// TIA Portal V18 export
FUNCTION "Operator message 2" : Void   // FC33, LAD
{ S7_Optimized_Access := 'TRUE' }
VERSION : 0.1
// stored: AutoNumber true, IsIECCheckEnabled false, SetENOAutomatically false, UDAEnableTagReadback false
BEGIN

REGION Network 1 (SCL)
   IF "Faults&warnings"."Critical Alarm Metering A" OR "Faults&warnings"."Critical Alarm metering B" OR "Faults&warnings"."Critical Alarm metering A&B" THEN
       "Faults&warnings"."Operator message 2" := 8; // Machine error
   ELSIF "Functions"."stop dosing function site" THEN
       "Faults&warnings"."Operator message 2" := 7; // Metering blocked
   ELSIF "Functions"."Dosing function selected" AND
       ("Faults&warnings"."Critical Alarm Metering A" OR "Faults&warnings"."Critical Alarm metering B" OR "Faults&warnings"."Critical Alarm metering A&B") THEN
       "Faults&warnings"."Operator message 2" := 6; // Metering blocked
   ELSIF "Functions"."Dosing function selected" AND "Functions"."Dosing Running" AND "Function_Selection_HMI"."Snuffback selected" AND
       ("Function_Selection_HMI".Function_Snuffback_volume_dispensed < "Function_Selection_HMI".Snuffback_qty) THEN
       "Faults&warnings"."Operator message 2" := 9;
   ELSIF "Functions"."Dosing function selected" AND "Functions"."Dosing Running" AND NOT ("Function_Selection_HMI"."Snuffback selected") THEN
       "Faults&warnings"."Operator message 2" := 5; //function running
   ELSIF "Control"."waiting For pre run" AND NOT ("Functions"."Dosing function selected") THEN
       "Faults&warnings"."Operator message 2" := 4; // waiting for prerun   
   ELSIF "Functions"."Dosing function selected" AND NOT ("Pump & Flowrate".startSnuff_Back_PumpA) AND NOT ("Pump & Flowrate".startSnuff_Back_PumpB) THEN
       "Faults&warnings"."Operator message 2" := 3; // waiting for start\
   ELSIF "Control"."waiting For pre run" = false THEN
       "Faults&warnings"."Operator message 2" := 2; // ready for operation
   ELSIF     "Faults&warnings"."Fault present" = false THEN
       "Faults&warnings"."Operator message 2" := 1; // machnie ready

   END_IF;
END_REGION
END_FUNCTION
